Fanuc KAREL source: ka00053.KL

-- PROVISIONAL review KL for V940-1; original PC SHA256 8f74b4d9ac7398b9338f013f4d3790915d61da4e41fdc2368a5daf647641c997
-- Incomplete behavior may be omitted. Consult companion uncertainty JSON. Do not deploy.
PROGRAM KA00053
%NOLOCKGROUP
-- UNRESOLVED_DECL SRC type=000101
-- UNRESOLVED_DECL DST type=000101
BEGIN
  -- V9_ZERO_TABLE_METADATA_HINT layout=0001; no indexed target words; source/name/runtime held
  -- UNRESOLVED_PC offsets 5-20; opcodes 49,4A
  -- UNRESOLVED_PC offsets 25-29; opcodes 7F
END KA00053
